// TIA Portal V19 export
DATA_BLOCK "A0302_Spintore"   // DB109
// stored: InstanceOfName A0302_Spintore_FB, InstanceOfType FB
"A0302_Spintore_FB"
   // VAR_INPUT
   //    AreaInterface : "AreaInterface";
   //    ZSI : "udt_ZoneSafetyInterface";
   //    DSI_Feed : "udt_DeviceSafetyInterface";
   //    DSI_Valve : "udt_DeviceSafetyInterface";
   //    Drive : "TAx_DriveInterface";
   //    DataIn : Struct
   //       OP : "OP_PB";
   //       P5 { ExternalAccessible := 'False'; ExternalVisible := 'False'; ExternalWritable := 'False'} : Struct
   //          Orz_AnalSens : Int;
   //          FTC_FuoriIngombro_A0301 : Bool;
   //       END_STRUCT;
   //    END_STRUCT;
   //    Cin : Struct
   //       Manager { ExternalWritable := 'False'} : Struct
   //          EnableStopDoorOpeningReq : Bool;
   //          EnableStopInPhase : Bool;
   //          EnableStopProgrammed : Bool;
   //          Control_ON : Bool;
   //          REST_Req : Bool;
   //          WORK_Req : Bool;
   //          Rest : Bool;
   //          Work : Bool;
   //       END_STRUCT;
   //       SemiAut_Pb { ExternalAccessible := 'False'; ExternalVisible := 'False'; ExternalWritable := 'False'} : Bool;
   //       P4 { ExternalWritable := 'False'} : Struct
   //          Fermi : "ValveMachine_COut";
   //       END_STRUCT;
   //       P5 { ExternalWritable := 'False'} : Struct
   //          "En/Dis_SpinLat_2" : Bool;
   //          QuotaIngombro_SpinLat2 : Real;
   //          QuotaIngombro_SpinLat1 : Real;
   //          Spintore_Lat : Struct
   //             Spin_Lat1 : Struct
   //                Standstill : Bool;
   //                Rest_CheckNext : Bool;
   //                Work_CheckNext : Bool;
   //                Rest : Bool;
   //                Work : Bool;
   //             END_STRUCT;
   //             Spin_Lat2 : Struct
   //                Standstill : Bool;
   //                Rest_CheckNext : Bool;
   //                Work_CheckNext : Bool;
   //                Rest : Bool;
   //                Work : Bool;
   //             END_STRUCT;
   //             Vrt_1 : "ValveMachine_COut";
   //             Orz_1 : "ValveMachine_COut";
   //             Vrt_2 : "ValveMachine_COut";
   //             Orz_2 : "ValveMachine_COut";
   //             Sollevatori : "ValveMachine_COut";
   //          END_STRUCT;
   //       END_STRUCT;
   //       Trasporto { ExternalAccessible := 'False'; ExternalVisible := 'False'; ExternalWritable := 'False'} : "SpeedMachine_COut";
   //       Bordatrice : Struct
   //          Ax : "Positioning_EPOS_Machine_COut";
   //          TargetVel : LReal;
   //          Perc_Vel : LReal;
   //          Sens : Struct
   //             FTC_Uscita : Bool;
   //          END_STRUCT;
   //       END_STRUCT;
   //    END_STRUCT;
   //    Config : Struct
   //       Ax : "Positioning_EPOS_Machine_Config_NEW";
   //       Vrt : "ValveMachine_Config";
   //       Orz : "ValveMachine_Config";
   //       SpintoreLat : Struct
   //          QuotaIngombro_SpinLat2 : Real;
   //          QuotaIngombro_SpinLat1 : Real;
   //       END_STRUCT;
   //       Bordatrice : Struct
   //          QuotaIngresso : Real;
   //       END_STRUCT;
   //       DelayMissingCondition : Time;
   //    END_STRUCT;
   //    HWID_Ax_TEL111 : HW_SUBMODULE;
   // END_VAR
   // VAR_OUTPUT
   //    MachineInterface : "MachineInterface";
   //    DataOut : "Positioning_EPOS_Machine_DataOut";
   //    COut : Struct
   //       Ax_Sts : Struct
   //          PosAttesa_Reached : Bool;
   //          PosFineSpinta_Reached : Bool;
   //       END_STRUCT;
   //       Ax : "Positioning_EPOS_Machine_COut";
   //       Spintore : "ValveMachine_COut";
   //       Vrt : "ValveMachine_COut";
   //       Orz : "ValveMachine_COut";
   //    END_STRUCT;
   // END_VAR
   // VAR_IN_OUT
   //    Par : Struct
   //       Sens : "Analogic_SensorManagement_Par";
   //    END_STRUCT;
   //    Data : Struct
   //       Sens : "Analogic_SensorManagement_Data";
   //       HMI : "HMI_Preset";
   //       Ax_Pos : "A0301_Mach_Ax_Pos_Data";
   //    END_STRUCT;
   //    Par_Mach : "A0301_Mach_Sens_Par";
   //    Par_Ax_Manu : "Positioning_EPOS_Machine_Par";
   //    Pers_Data : Struct
   //       EncoderAbsolute_Preset_OK : Bool;
   //       Persistent_ActualPosition : LReal;
   //    END_STRUCT;
   //    Par_Ax_Auto : "A0301_Mach_Speed_Par";
   // END_VAR
   // VAR
   //    Alarm : Struct
   //       Ax : "Positioning_EPOS_Machine_Alr";
   //       Ax_NeedPreset { S7_SetPoint := 'True'} : Bool;
   //       Vrt : "ValveAlr";
   //       Orz : "ValveAlr";
   //       Orz_AnalSens_Issue : Bool;
   //       Orz_AnalSens_Compressed : Bool;
   //    END_STRUCT;
   //    Warning : Struct
   //       Ax : "Positioning_EPOS_Machine_Wng";
   //       Vrt : "ValveMachine_Wng";
   //       Orz { S7_SetPoint := 'True'} : "ValveMachine_Wng";
   //       Orz_AnalSens { S7_SetPoint := 'True'} : "Analogic_SensorManagement_Warning";
   //       OP_REST_MissingCnd : Bool;
   //       OP_WORK_MissingCnd : Bool;
   //    END_STRUCT;
   //    Sts : Struct
   //       ReadyForMove : Bool;
   //       OP_CanMoveFreely : Bool;
   //       OP_Ax_Rest_Cnd : Bool;
   //       OP_Ax_Work_Cnd : Bool;
   //       OP_Spin_Rest_Cnd : Bool;
   //       OP_Spin_Work_Cnd : Bool;
   //       A0301_Beam_BLean : Real;
   //       A0302_Beam_BLean : Real;
   //       Vrt_Work_ExtEnable : Bool;
   //       Orz_Work_ExtEnable : Bool;
   //    END_STRUCT;
   //    Ctrl : Struct
   //       SpinVrtOrz : Struct
   //          OP_Rest_Man : Bool;
   //          OP_Work_Man : Bool;
   //          OP_Rest_Aut : Bool;
   //          OP_Work_Aut : Bool;
   //          OP_Rest : Bool;
   //          OP_Work : Bool;
   //       END_STRUCT;
   //       Ax : Struct
   //          OP_Rest_Man : Bool;
   //          OP_Work_Man : Bool;
   //          OP_Rest_Aut : Bool;
   //          OP_Work_Aut : Bool;
   //          OP_Rest : Bool;
   //          OP_Work : Bool;
   //          Vel : LReal;
   //          VelMax : Real;
   //          Dec : LReal;
   //       END_STRUCT;
   //    END_STRUCT;
   //    HMI : Struct
   //       Ax : "AnalogSens_HmiData";
   //       Orz_AnalSens_PB_Preset { ExternalAccessible := 'False'; ExternalVisible := 'False'; ExternalWritable := 'False'} : Bool;
   //       Orz_AnalSens_Preset_Value : LReal;
   //    END_STRUCT;
   //    Ax { S7_SetPoint := 'True'} : "Positioning_EPOS_Machine_FB_NEW";
   //    Vrt { S7_SetPoint := 'True'} : "ValveMachine_FB";
   //    Orz { S7_SetPoint := 'True'} : "ValveMachine_FB";
   //    Orz_AnalSens { S7_SetPoint := 'True'} : "Analogic_SensorManagement";
   //    ValueBLeanOvr : Array[1..15] of Real;
   //    IEC : Struct
   //       TON_DelayFTC_Ingombro_A0301 : IEC_TIMER;
   //       TOF_DelayFTC_Ingombro_A0301 { S7_SetPoint := 'True'} : IEC_TIMER;
   //       FTC_On { S7_SetPoint := 'True'} : Bool;
   //    END_STRUCT;
   //    AUX : Struct
   //       OP_Rest_PB : Bool;
   //       OP_Work_PB : Bool;
   //    END_STRUCT;
   //    TON_OP_REST_MissingCnd { S7_SetPoint := 'True'} : TON_TIME;
   //    TON_OP_WORK_MissingCnd { S7_SetPoint := 'True'} : TON_TIME;
   //    BTrk_Item : Struct
   //       BLean : Real;
   //       O_ID : DInt;
   //    END_STRUCT;
   // END_VAR
BEGIN
END_DATA_BLOCK
